PROGRAM MAIN
VAR
END_VAR

//First GIT

END_PROGRAM

(* stored: Version 1.1.0.1, ProductVersion 3.1.4024.11
   POU MAIN: Id {8679e355-f72d-448c-a2ed-9730846f6a1f}, SpecialFunc None *)
